FUNCTION_BLOCK Assembly_Conveyor
VAR_INPUT
	cmdRunFwd 			: BOOL;
	cmdRunRev 			: BOOL;
	cmdStop 			: BOOL;
	cfgRestartDelay		: TIME;
	inpTensionOK AT %I*	: BOOL;
END_VAR
VAR_OUTPUT
END_VAR
VAR
END_VAR

END_FUNCTION_BLOCK

(* stored: Version 1.1.0.1, ProductVersion 3.1.4022.11
   POU Assembly_Conveyor: Id {d460b149-adbf-4df5-9d39-6f1da505c84e}, SpecialFunc None *)
